FUNCTION FlowOut : REAL

VAR
	a : REAL := 14 * EXPT(10,-4);
	b : REAL := GVL.valve_oule;
	c : REAL := SQRT(2 * GVL.const_grav * GVL.high_now);
END_VAR

GVL.flow_out := a * b * c;
FlowOut :=  GVL.flow_out;

END_FUNCTION

(* stored: Version 1.1.0.1, ProductVersion 3.1.4024.12
   POU FlowOut: Id {9eb8b10c-54cd-4142-b2a4-1aa0751dd7b0}, SpecialFunc None *)
